// TIA Portal V19 export
TYPE "ValveMachine_DataOut"
// stored: Access Published
   STRUCT
      RestSolenoid : Bool;
      WorkSolenoid : Bool;
   END_STRUCT;
END_TYPE
